// Mitsubishi GX Works2 project: 视觉检测   PLC: FX3S

PROGRAM MAIN
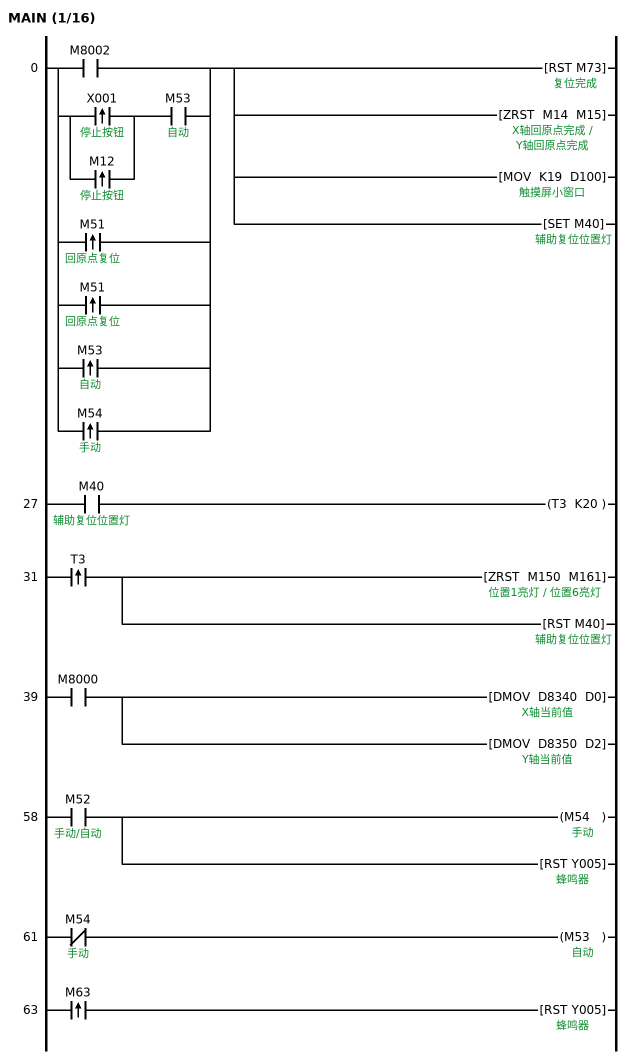
0     LD      M8002
      LDP     X001  ; 停止按钮
      ORP     M12  ; 停止按钮
      AND     M53  ; 自动
      ORB
      ORP     M51  ; 回原点复位
      ORP     M51  ; 回原点复位
      ORP     M53  ; 自动
      ORP     M54  ; 手动
      RST     M73  ; 复位完成
      ZRST    M14 M15  ; X轴回原点完成 / Y轴回原点完成
      MOV     K19 D100  ; 触摸屏小窗口
      SET     M40  ; 辅助复位位置灯
27    LD      M40  ; 辅助复位位置灯
      OUT     T3 K20
31    LDP     T3
      ZRST    M150 M161  ; 位置1亮灯 / 位置6亮灯
      RST     M40  ; 辅助复位位置灯
39    LD      M8000
      DMOV    D8340 D0  ; X轴当前值
      DMOV    D8350 D2  ; Y轴当前值
58    LD      M52  ; 手动/自动
      OUT     M54  ; 手动
      RST     Y005  ; 蜂鸣器
61    LDI     M54  ; 手动
      OUT     M53  ; 自动
63    LDP     M63
      RST     Y005  ; 蜂鸣器
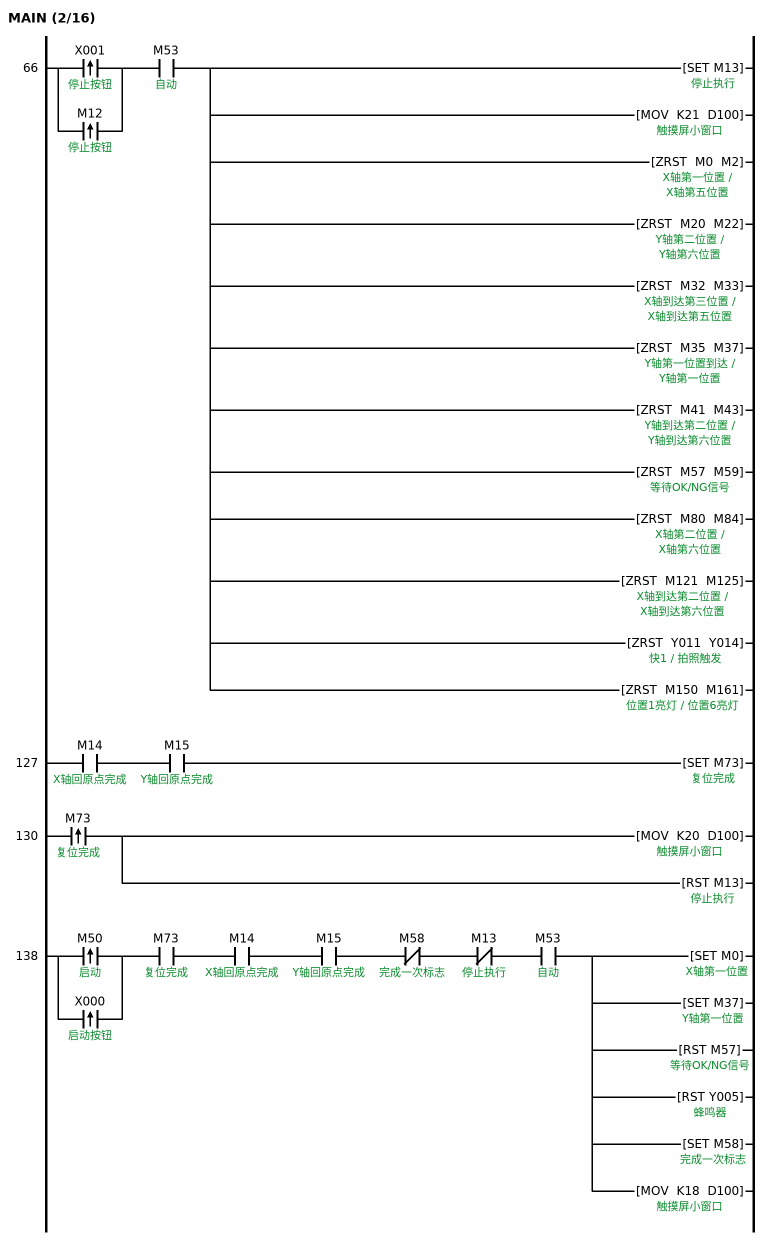
66    LDP     X001  ; 停止按钮
      ORP     M12  ; 停止按钮
      AND     M53  ; 自动
      SET     M13  ; 停止执行
      MOV     K21 D100
      ZRST    M0 M2  ; X轴第一位置 / X轴第五位置
      ZRST    M20 M22  ; Y轴第二位置 / Y轴第六位置
      ZRST    M32 M33  ; X轴到达第三位置 / X轴到达第五位置
      ZRST    M35 M37  ; Y轴第一位置到达 / Y轴第一位置
      ZRST    M41 M43  ; Y轴到达第二位置 / Y轴到达第六位置
      ZRST    M57 M59  ; 等待OK/NG信号
      ZRST    M80 M84  ; X轴第二位置 / X轴第六位置
      ZRST    M121 M125  ; X轴到达第二位置 / X轴到达第六位置
      ZRST    Y011 Y014  ; 快1 / 拍照触发
      ZRST    M150 M161
127   LD      M14  ; X轴回原点完成
      AND     M15  ; Y轴回原点完成
      SET     M73  ; 复位完成
130   LDP     M73  ; 复位完成
      MOV     K20 D100
      RST     M13  ; 停止执行
138   LDP     M50  ; 启动
      ORP     X000  ; 启动按钮
      AND     M73  ; 复位完成
      AND     M14  ; X轴回原点完成
      AND     M15  ; Y轴回原点完成
      ANI     M58  ; 完成一次标志
      ANI     M13  ; 停止执行
      AND     M53  ; 自动
      SET     M0  ; X轴第一位置
      SET     M37  ; Y轴第一位置
      RST     M57  ; 等待OK/NG信号
      RST     Y005  ; 蜂鸣器
      SET     M58  ; 完成一次标志
      MOV     K18 D100
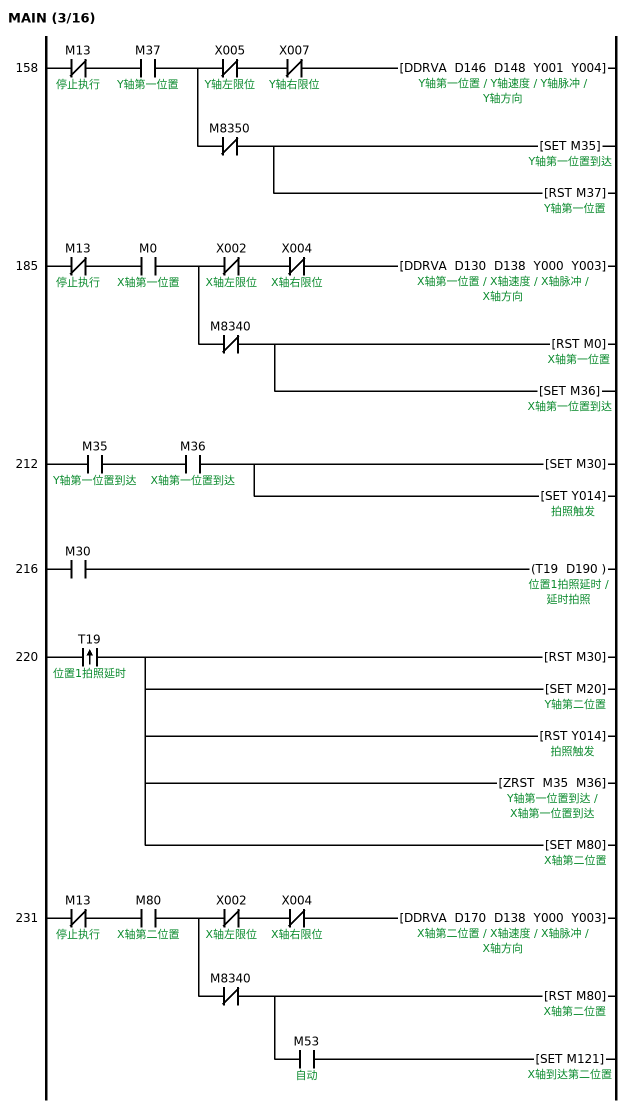
158   LDI     M13  ; 停止执行
      AND     M37  ; Y轴第一位置
      MPS
      ANI     X005  ; Y轴左限位
      ANI     X007  ; Y轴右限位
      DDRVA   D146 D148 Y001 Y004  ; Y轴第一位置 / Y轴速度 / Y轴脉冲 / Y轴方向
      MPP
      ANI     M8350
      SET     M35  ; Y轴第一位置到达
      RST     M37  ; Y轴第一位置
185   LDI     M13  ; 停止执行
      AND     M0  ; X轴第一位置
      MPS
      ANI     X002  ; X轴左限位
      ANI     X004  ; X轴右限位
      DDRVA   D130 D138 Y000 Y003  ; X轴第一位置 / X轴速度 / X轴脉冲 / X轴方向
      MPP
      ANI     M8340
      RST     M0  ; X轴第一位置
      SET     M36  ; X轴第一位置到达
212   LD      M35  ; Y轴第一位置到达
      AND     M36  ; X轴第一位置到达
      SET     M30
      SET     Y014  ; 拍照触发
216   LD      M30
      OUT     T19 D190  ; 位置1拍照延时 / 延时拍照
220   LDP     T19  ; 位置1拍照延时
      RST     M30
      SET     M20  ; Y轴第二位置
      RST     Y014  ; 拍照触发
      ZRST    M35 M36
      SET     M80  ; X轴第二位置
231   LDI     M13  ; 停止执行
      AND     M80  ; X轴第二位置
      MPS
      ANI     X002  ; X轴左限位
      ANI     X004  ; X轴右限位
      DDRVA   D170 D138 Y000 Y003  ; X轴第二位置
      MPP
      ANI     M8340
      RST     M80  ; X轴第二位置
      AND     M53  ; 自动
      SET     M121  ; X轴到达第二位置
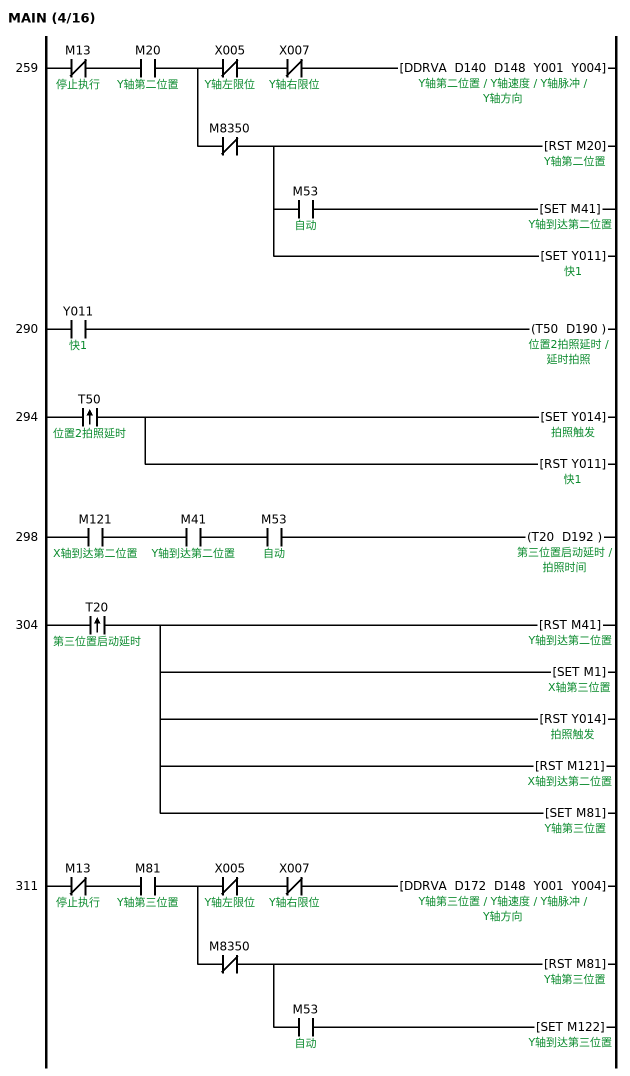
259   LDI     M13  ; 停止执行
      AND     M20  ; Y轴第二位置
      MPS
      ANI     X005  ; Y轴左限位
      ANI     X007  ; Y轴右限位
      DDRVA   D140 D148 Y001 Y004  ; Y轴第二位置
      MPP
      ANI     M8350
      RST     M20  ; Y轴第二位置
      MPS
      AND     M53  ; 自动
      SET     M41  ; Y轴到达第二位置
      MPP
      SET     Y011  ; 快1
290   LD      Y011  ; 快1
      OUT     T50 D190  ; 位置2拍照延时 / 延时拍照
294   LDP     T50  ; 位置2拍照延时
      SET     Y014  ; 拍照触发
      RST     Y011  ; 快1
298   LD      M121  ; X轴到达第二位置
      AND     M41  ; Y轴到达第二位置
      AND     M53  ; 自动
      OUT     T20 D192  ; 第三位置启动延时 / 拍照时间
304   LDP     T20  ; 第三位置启动延时
      RST     M41  ; Y轴到达第二位置
      SET     M1  ; X轴第三位置
      RST     Y014  ; 拍照触发
      RST     M121  ; X轴到达第二位置
      SET     M81  ; Y轴第三位置
311   LDI     M13  ; 停止执行
      AND     M81  ; Y轴第三位置
      MPS
      ANI     X005  ; Y轴左限位
      ANI     X007  ; Y轴右限位
      DDRVA   D172 D148 Y001 Y004  ; Y轴第三位置
      MPP
      ANI     M8350
      RST     M81  ; Y轴第三位置
      AND     M53  ; 自动
      SET     M122  ; Y轴到达第三位置
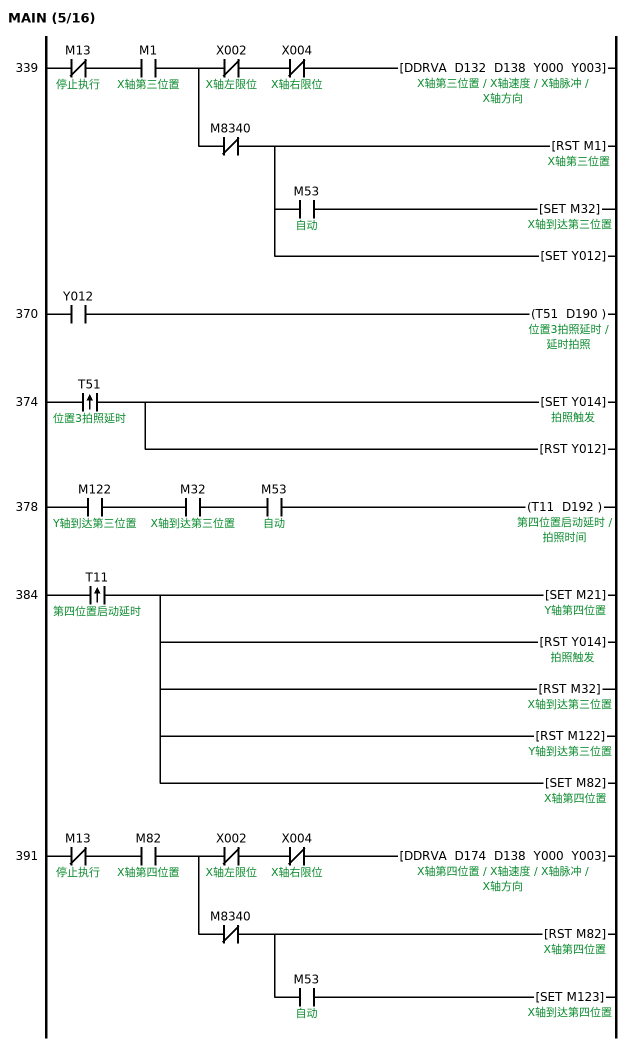
339   LDI     M13  ; 停止执行
      AND     M1  ; X轴第三位置
      MPS
      ANI     X002  ; X轴左限位
      ANI     X004  ; X轴右限位
      DDRVA   D132 D138 Y000 Y003  ; X轴第三位置
      MPP
      ANI     M8340
      RST     M1  ; X轴第三位置
      MPS
      AND     M53  ; 自动
      SET     M32  ; X轴到达第三位置
      MPP
      SET     Y012
370   LD      Y012
      OUT     T51 D190  ; 位置3拍照延时 / 延时拍照
374   LDP     T51  ; 位置3拍照延时
      SET     Y014  ; 拍照触发
      RST     Y012
378   LD      M122  ; Y轴到达第三位置
      AND     M32  ; X轴到达第三位置
      AND     M53  ; 自动
      OUT     T11 D192  ; 第四位置启动延时 / 拍照时间
384   LDP     T11  ; 第四位置启动延时
      SET     M21  ; Y轴第四位置
      RST     Y014  ; 拍照触发
      RST     M32  ; X轴到达第三位置
      RST     M122  ; Y轴到达第三位置
      SET     M82  ; X轴第四位置
391   LDI     M13  ; 停止执行
      AND     M82  ; X轴第四位置
      MPS
      ANI     X002  ; X轴左限位
      ANI     X004  ; X轴右限位
      DDRVA   D174 D138 Y000 Y003  ; X轴第四位置
      MPP
      ANI     M8340
      RST     M82  ; X轴第四位置
      AND     M53  ; 自动
      SET     M123  ; X轴到达第四位置
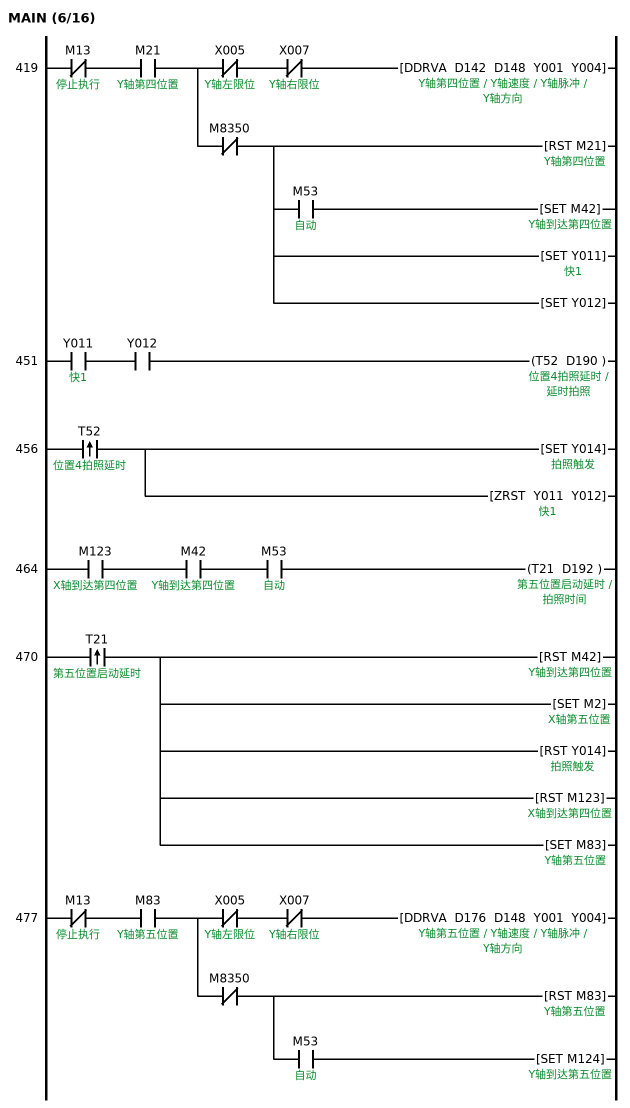
419   LDI     M13  ; 停止执行
      AND     M21  ; Y轴第四位置
      MPS
      ANI     X005  ; Y轴左限位
      ANI     X007  ; Y轴右限位
      DDRVA   D142 D148 Y001 Y004  ; Y轴第四位置
      MPP
      ANI     M8350
      RST     M21  ; Y轴第四位置
      MPS
      AND     M53  ; 自动
      SET     M42  ; Y轴到达第四位置
      MPP
      SET     Y011  ; 快1
      SET     Y012
451   LD      Y011  ; 快1
      AND     Y012
      OUT     T52 D190  ; 位置4拍照延时 / 延时拍照
456   LDP     T52  ; 位置4拍照延时
      SET     Y014  ; 拍照触发
      ZRST    Y011 Y012
464   LD      M123  ; X轴到达第四位置
      AND     M42  ; Y轴到达第四位置
      AND     M53  ; 自动
      OUT     T21 D192  ; 第五位置启动延时 / 拍照时间
470   LDP     T21  ; 第五位置启动延时
      RST     M42  ; Y轴到达第四位置
      SET     M2  ; X轴第五位置
      RST     Y014  ; 拍照触发
      RST     M123  ; X轴到达第四位置
      SET     M83  ; Y轴第五位置
477   LDI     M13  ; 停止执行
      AND     M83  ; Y轴第五位置
      MPS
      ANI     X005  ; Y轴左限位
      ANI     X007  ; Y轴右限位
      DDRVA   D176 D148 Y001 Y004  ; Y轴第五位置
      MPP
      ANI     M8350
      RST     M83  ; Y轴第五位置
      AND     M53  ; 自动
      SET     M124  ; Y轴到达第五位置
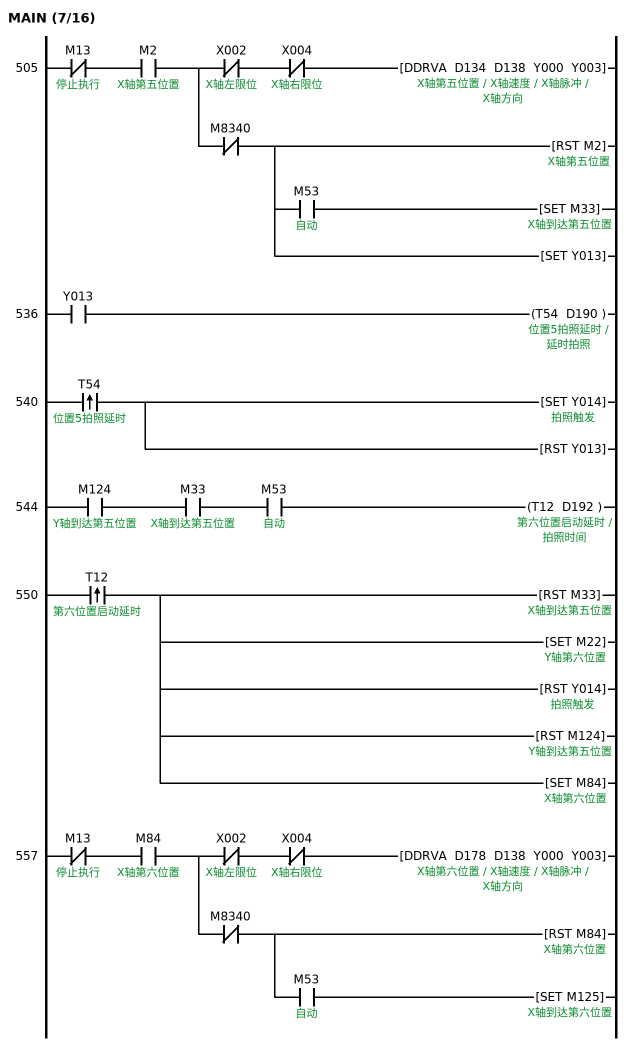
505   LDI     M13  ; 停止执行
      AND     M2  ; X轴第五位置
      MPS
      ANI     X002  ; X轴左限位
      ANI     X004  ; X轴右限位
      DDRVA   D134 D138 Y000 Y003  ; X轴第五位置
      MPP
      ANI     M8340
      RST     M2  ; X轴第五位置
      MPS
      AND     M53  ; 自动
      SET     M33  ; X轴到达第五位置
      MPP
      SET     Y013
536   LD      Y013
      OUT     T54 D190  ; 位置5拍照延时 / 延时拍照
540   LDP     T54  ; 位置5拍照延时
      SET     Y014  ; 拍照触发
      RST     Y013
544   LD      M124  ; Y轴到达第五位置
      AND     M33  ; X轴到达第五位置
      AND     M53  ; 自动
      OUT     T12 D192  ; 第六位置启动延时 / 拍照时间
550   LDP     T12  ; 第六位置启动延时
      RST     M33  ; X轴到达第五位置
      SET     M22  ; Y轴第六位置
      RST     Y014  ; 拍照触发
      RST     M124  ; Y轴到达第五位置
      SET     M84  ; X轴第六位置
557   LDI     M13  ; 停止执行
      AND     M84  ; X轴第六位置
      MPS
      ANI     X002  ; X轴左限位
      ANI     X004  ; X轴右限位
      DDRVA   D178 D138 Y000 Y003  ; X轴第六位置
      MPP
      ANI     M8340
      RST     M84  ; X轴第六位置
      AND     M53  ; 自动
      SET     M125  ; X轴到达第六位置
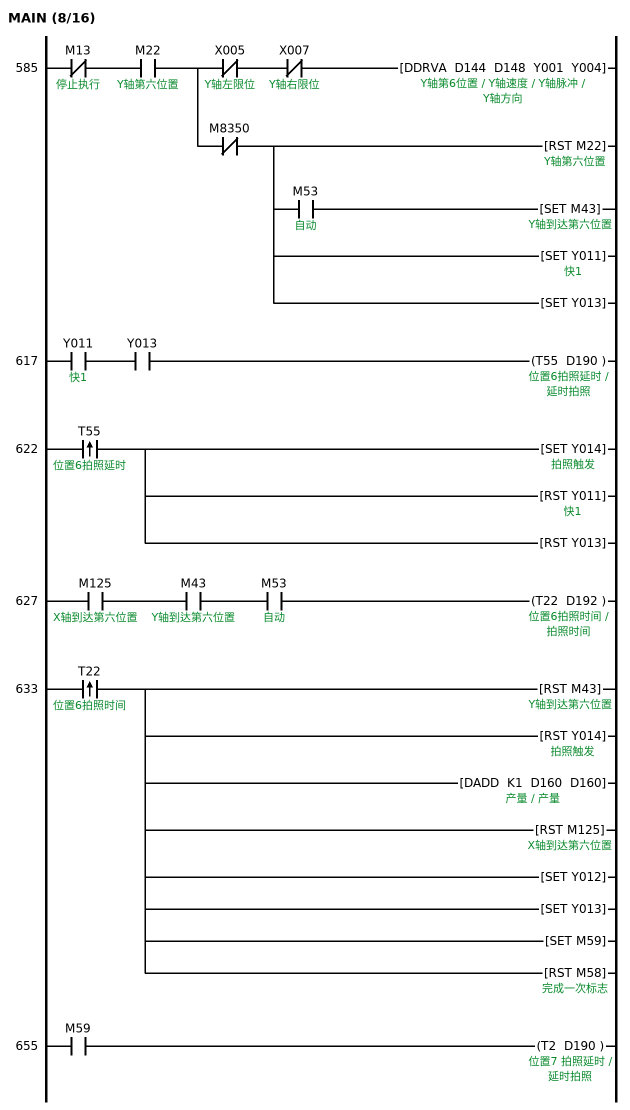
585   LDI     M13  ; 停止执行
      AND     M22  ; Y轴第六位置
      MPS
      ANI     X005  ; Y轴左限位
      ANI     X007  ; Y轴右限位
      DDRVA   D144 D148 Y001 Y004  ; Y轴第6位置
      MPP
      ANI     M8350
      RST     M22  ; Y轴第六位置
      MPS
      AND     M53  ; 自动
      SET     M43  ; Y轴到达第六位置
      MPP
      SET     Y011  ; 快1
      SET     Y013
617   LD      Y011  ; 快1
      AND     Y013
      OUT     T55 D190  ; 位置6拍照延时 / 延时拍照
622   LDP     T55  ; 位置6拍照延时
      SET     Y014  ; 拍照触发
      RST     Y011  ; 快1
      RST     Y013
627   LD      M125  ; X轴到达第六位置
      AND     M43  ; Y轴到达第六位置
      AND     M53  ; 自动
      OUT     T22 D192  ; 位置6拍照时间 / 拍照时间
633   LDP     T22  ; 位置6拍照时间
      RST     M43  ; Y轴到达第六位置
      RST     Y014  ; 拍照触发
      DADD    K1 D160 D160  ; 产量
      RST     M125  ; X轴到达第六位置
      SET     Y012
      SET     Y013
      SET     M59
      RST     M58  ; 完成一次标志
655   LD      M59
      OUT     T2 D190  ; 位置7 拍照延时 / 延时拍照
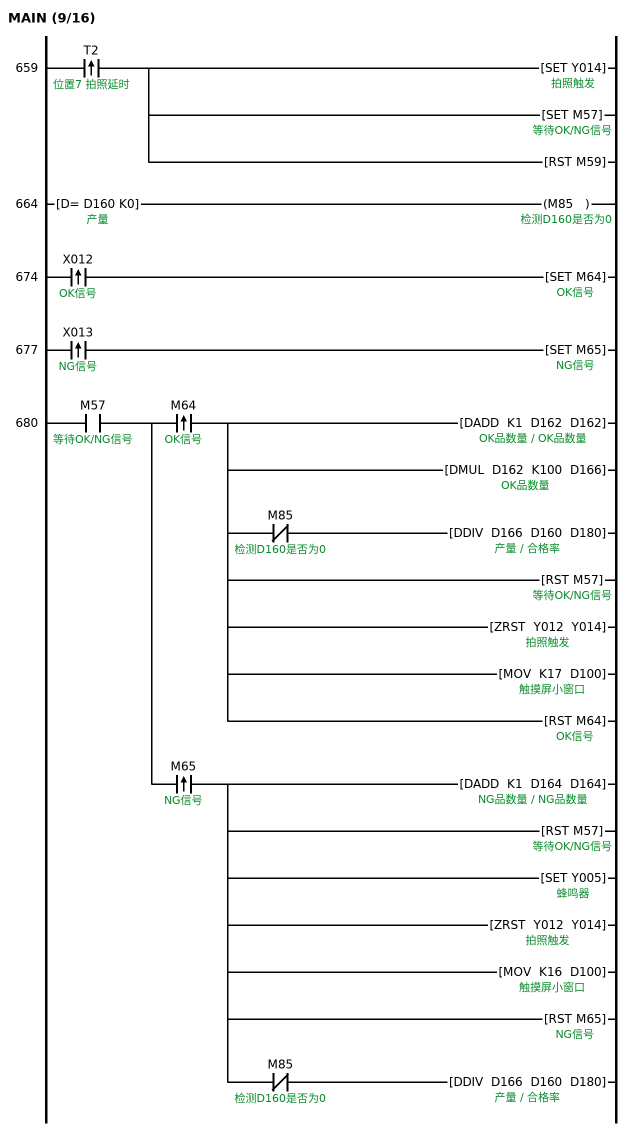
659   LDP     T2  ; 位置7 拍照延时
      SET     Y014  ; 拍照触发
      SET     M57  ; 等待OK/NG信号
      RST     M59
664   LDD=    D160 K0  ; 产量
      OUT     M85  ; 检测D160是否为0
674   LDP     X012  ; OK信号
      SET     M64  ; OK信号
677   LDP     X013  ; NG信号
      SET     M65  ; NG信号
680   LD      M57  ; 等待OK/NG信号
      MPS
      ANDP    M64  ; OK信号
      DADD    K1 D162 D162  ; OK品数量
      DMUL    D162 K100 D166
      MPS
      ANI     M85  ; 检测D160是否为0
      DDIV    D166 D160 D180  ; 合格率
      MPP
      RST     M57  ; 等待OK/NG信号
      ZRST    Y012 Y014
      MOV     K17 D100
      RST     M64  ; OK信号
      MPP
      ANDP    M65  ; NG信号
      DADD    K1 D164 D164  ; NG品数量
      RST     M57  ; 等待OK/NG信号
      SET     Y005  ; 蜂鸣器
      ZRST    Y012 Y014
      MOV     K16 D100
      RST     M65  ; NG信号
      ANI     M85  ; 检测D160是否为0
      DDIV    D166 D160 D180
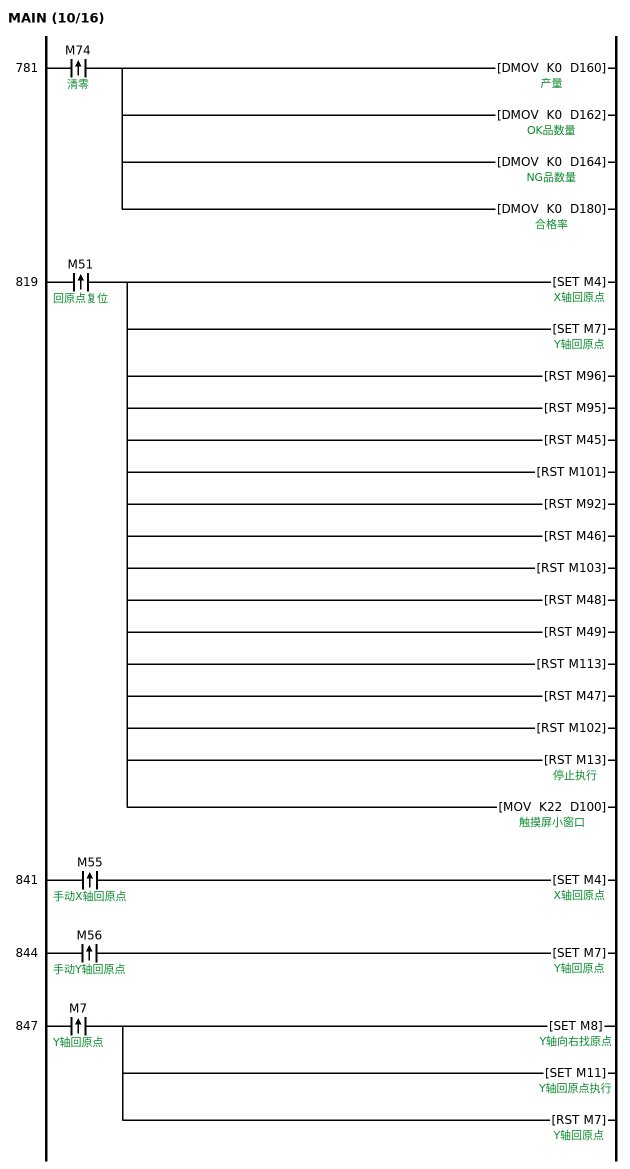
781   LDP     M74  ; 清零
      DMOV    K0 D160
      DMOV    K0 D162
      DMOV    K0 D164
      DMOV    K0 D180
819   LDP     M51  ; 回原点复位
      SET     M4  ; X轴回原点
      SET     M7  ; Y轴回原点
      RST     M96
      RST     M95
      RST     M45
      RST     M101
      RST     M92
      RST     M46
      RST     M103
      RST     M48
      RST     M49
      RST     M113
      RST     M47
      RST     M102
      RST     M13  ; 停止执行
      MOV     K22 D100
841   LDP     M55  ; 手动X轴回原点
      SET     M4  ; X轴回原点
844   LDP     M56  ; 手动Y轴回原点
      SET     M7  ; Y轴回原点
847   LDP     M7  ; Y轴回原点
      SET     M8  ; Y轴向右找原点
      SET     M11  ; Y轴回原点执行
      RST     M7  ; Y轴回原点
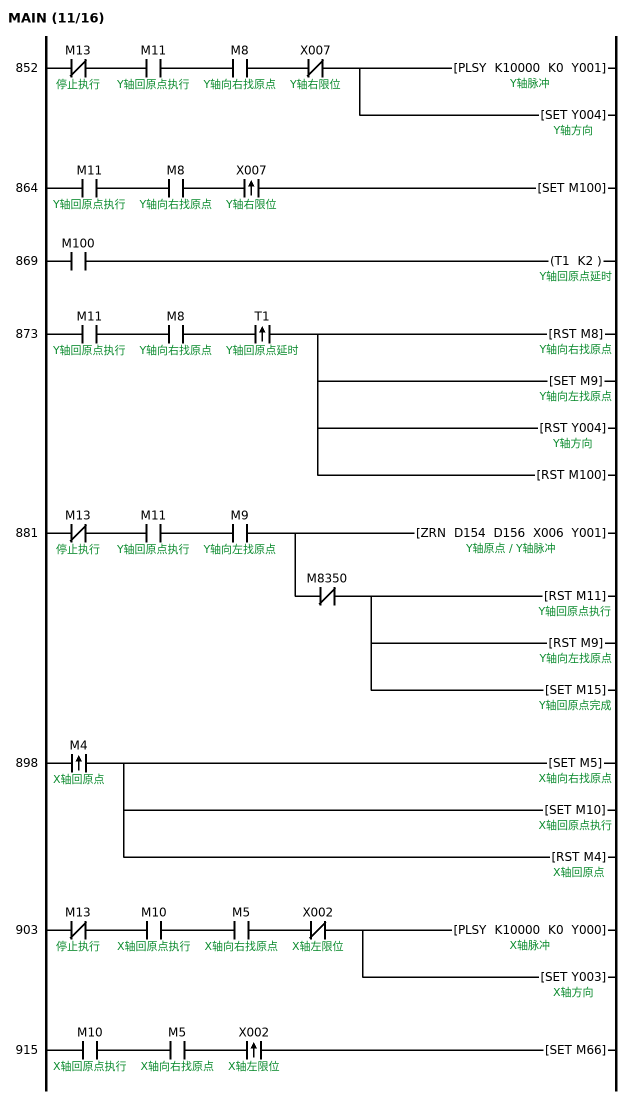
852   LDI     M13  ; 停止执行
      AND     M11  ; Y轴回原点执行
      AND     M8  ; Y轴向右找原点
      ANI     X007  ; Y轴右限位
      PLSY    K10000 K0 Y001  ; Y轴脉冲
      SET     Y004  ; Y轴方向
864   LD      M11  ; Y轴回原点执行
      AND     M8  ; Y轴向右找原点
      ANDP    X007  ; Y轴右限位
      SET     M100
869   LD      M100
      OUT     T1 K2  ; Y轴回原点延时
873   LD      M11  ; Y轴回原点执行
      AND     M8  ; Y轴向右找原点
      ANDP    T1  ; Y轴回原点延时
      RST     M8  ; Y轴向右找原点
      SET     M9  ; Y轴向左找原点
      RST     Y004  ; Y轴方向
      RST     M100
881   LDI     M13  ; 停止执行
      AND     M11  ; Y轴回原点执行
      AND     M9  ; Y轴向左找原点
      ZRN     D154 D156 X006 Y001  ; Y轴原点
      ANI     M8350
      RST     M11  ; Y轴回原点执行
      RST     M9  ; Y轴向左找原点
      SET     M15  ; Y轴回原点完成
898   LDP     M4  ; X轴回原点
      SET     M5  ; X轴向右找原点
      SET     M10  ; X轴回原点执行
      RST     M4  ; X轴回原点
903   LDI     M13  ; 停止执行
      AND     M10  ; X轴回原点执行
      AND     M5  ; X轴向右找原点
      ANI     X002  ; X轴左限位
      PLSY    K10000 K0 Y000  ; X轴脉冲
      SET     Y003  ; X轴方向
915   LD      M10  ; X轴回原点执行
      AND     M5  ; X轴向右找原点
      ANDP    X002  ; X轴左限位
      SET     M66
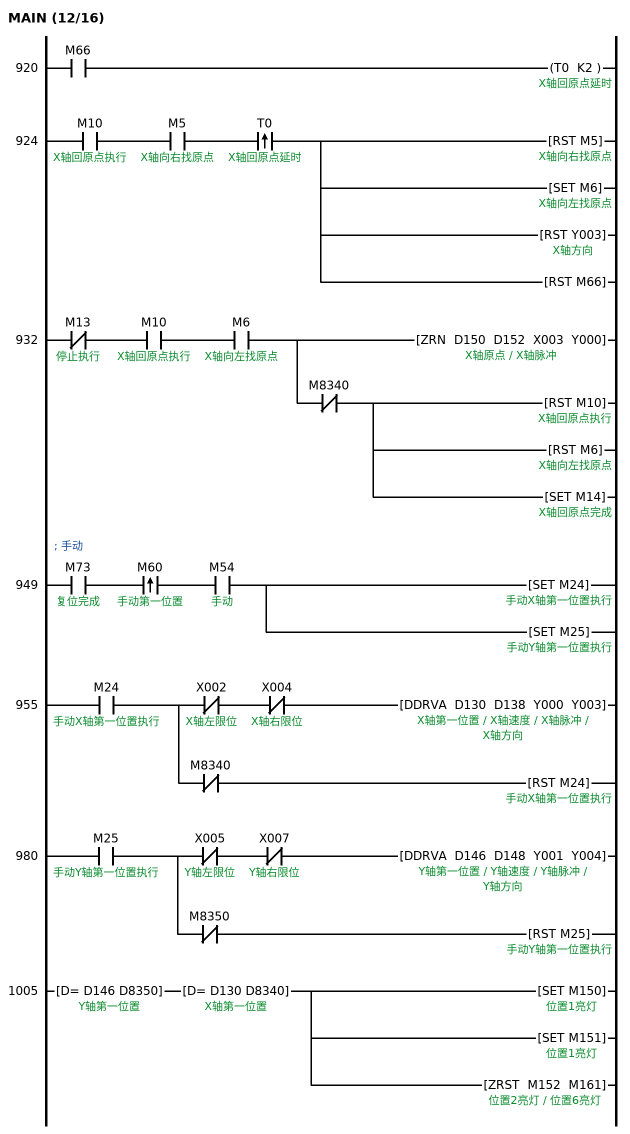
920   LD      M66
      OUT     T0 K2  ; X轴回原点延时
924   LD      M10  ; X轴回原点执行
      AND     M5  ; X轴向右找原点
      ANDP    T0  ; X轴回原点延时
      RST     M5  ; X轴向右找原点
      SET     M6  ; X轴向左找原点
      RST     Y003  ; X轴方向
      RST     M66
932   LDI     M13  ; 停止执行
      AND     M10  ; X轴回原点执行
      AND     M6  ; X轴向左找原点
      ZRN     D150 D152 X003 Y000  ; X轴原点
      ANI     M8340
      RST     M10  ; X轴回原点执行
      RST     M6  ; X轴向左找原点
      SET     M14  ; X轴回原点完成
; 手动
949   LD      M73  ; 复位完成
      ANDP    M60  ; 手动第一位置
      AND     M54  ; 手动
      SET     M24  ; 手动X轴第一位置执行
      SET     M25  ; 手动Y轴第一位置执行
955   LD      M24  ; 手动X轴第一位置执行
      MPS
      ANI     X002  ; X轴左限位
      ANI     X004  ; X轴右限位
      DDRVA   D130 D138 Y000 Y003
      MPP
      ANI     M8340
      RST     M24  ; 手动X轴第一位置执行
980   LD      M25  ; 手动Y轴第一位置执行
      MPS
      ANI     X005  ; Y轴左限位
      ANI     X007  ; Y轴右限位
      DDRVA   D146 D148 Y001 Y004
      MPP
      ANI     M8350
      RST     M25  ; 手动Y轴第一位置执行
1005  LDD=    D146 D8350  ; Y轴第一位置
      ANDD=   D130 D8340  ; X轴第一位置
      SET     M150  ; 位置1亮灯
      SET     M151  ; 位置1亮灯
      ZRST    M152 M161  ; 位置2亮灯
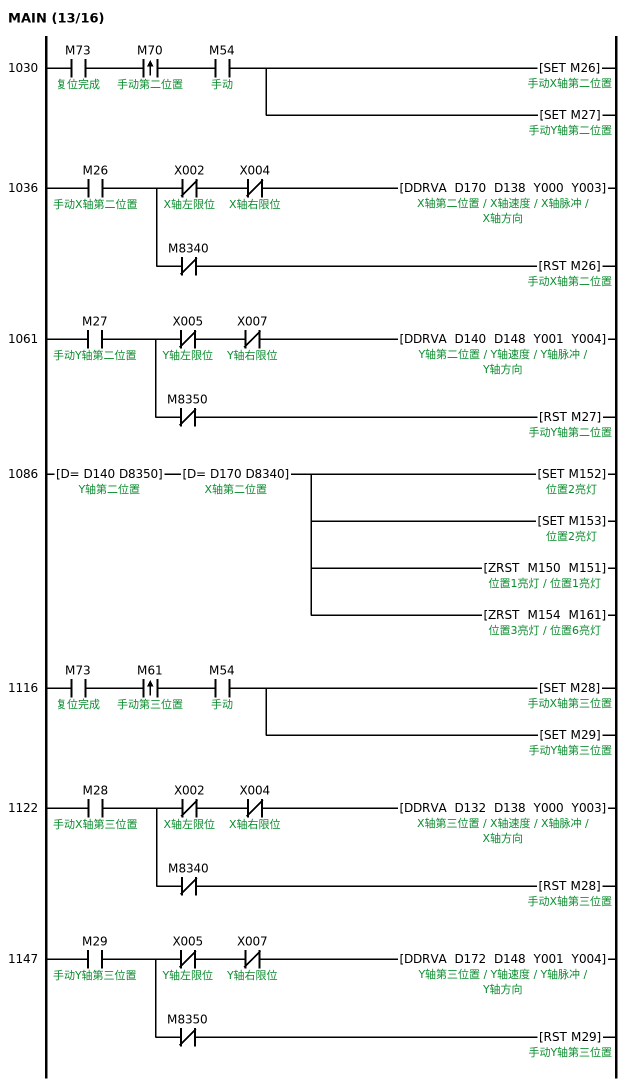
1030  LD      M73  ; 复位完成
      ANDP    M70  ; 手动第二位置
      AND     M54  ; 手动
      SET     M26  ; 手动X轴第二位置
      SET     M27  ; 手动Y轴第二位置
1036  LD      M26  ; 手动X轴第二位置
      MPS
      ANI     X002  ; X轴左限位
      ANI     X004  ; X轴右限位
      DDRVA   D170 D138 Y000 Y003
      MPP
      ANI     M8340
      RST     M26  ; 手动X轴第二位置
1061  LD      M27  ; 手动Y轴第二位置
      MPS
      ANI     X005  ; Y轴左限位
      ANI     X007  ; Y轴右限位
      DDRVA   D140 D148 Y001 Y004
      MPP
      ANI     M8350
      RST     M27  ; 手动Y轴第二位置
1086  LDD=    D140 D8350  ; Y轴第二位置
      ANDD=   D170 D8340  ; X轴第二位置
      SET     M152  ; 位置2亮灯
      SET     M153  ; 位置2亮灯
      ZRST    M150 M151
      ZRST    M154 M161  ; 位置3亮灯
1116  LD      M73  ; 复位完成
      ANDP    M61  ; 手动第三位置
      AND     M54  ; 手动
      SET     M28  ; 手动X轴第三位置
      SET     M29  ; 手动Y轴第三位置
1122  LD      M28  ; 手动X轴第三位置
      MPS
      ANI     X002  ; X轴左限位
      ANI     X004  ; X轴右限位
      DDRVA   D132 D138 Y000 Y003
      MPP
      ANI     M8340
      RST     M28  ; 手动X轴第三位置
1147  LD      M29  ; 手动Y轴第三位置
      MPS
      ANI     X005  ; Y轴左限位
      ANI     X007  ; Y轴右限位
      DDRVA   D172 D148 Y001 Y004
      MPP
      ANI     M8350
      RST     M29  ; 手动Y轴第三位置
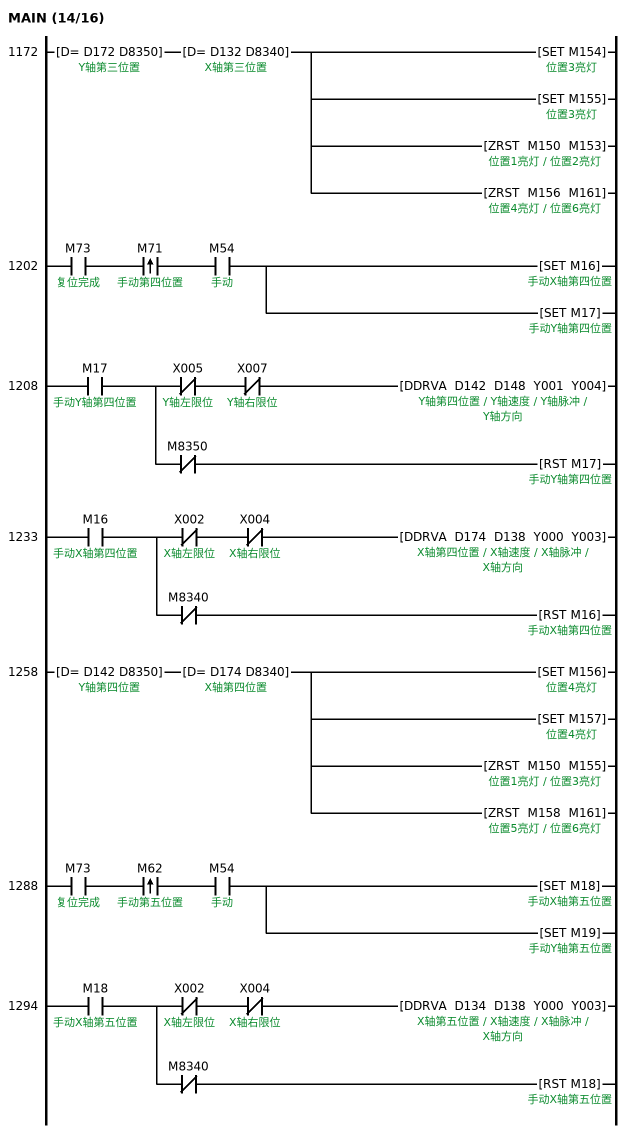
1172  LDD=    D172 D8350  ; Y轴第三位置
      ANDD=   D132 D8340  ; X轴第三位置
      SET     M154  ; 位置3亮灯
      SET     M155  ; 位置3亮灯
      ZRST    M150 M153
      ZRST    M156 M161  ; 位置4亮灯
1202  LD      M73  ; 复位完成
      ANDP    M71  ; 手动第四位置
      AND     M54  ; 手动
      SET     M16  ; 手动X轴第四位置
      SET     M17  ; 手动Y轴第四位置
1208  LD      M17  ; 手动Y轴第四位置
      MPS
      ANI     X005  ; Y轴左限位
      ANI     X007  ; Y轴右限位
      DDRVA   D142 D148 Y001 Y004
      MPP
      ANI     M8350
      RST     M17  ; 手动Y轴第四位置
1233  LD      M16  ; 手动X轴第四位置
      MPS
      ANI     X002  ; X轴左限位
      ANI     X004  ; X轴右限位
      DDRVA   D174 D138 Y000 Y003
      MPP
      ANI     M8340
      RST     M16  ; 手动X轴第四位置
1258  LDD=    D142 D8350  ; Y轴第四位置
      ANDD=   D174 D8340  ; X轴第四位置
      SET     M156  ; 位置4亮灯
      SET     M157  ; 位置4亮灯
      ZRST    M150 M155
      ZRST    M158 M161  ; 位置5亮灯
1288  LD      M73  ; 复位完成
      ANDP    M62  ; 手动第五位置
      AND     M54  ; 手动
      SET     M18  ; 手动X轴第五位置
      SET     M19  ; 手动Y轴第五位置
1294  LD      M18  ; 手动X轴第五位置
      MPS
      ANI     X002  ; X轴左限位
      ANI     X004  ; X轴右限位
      DDRVA   D134 D138 Y000 Y003
      MPP
      ANI     M8340
      RST     M18  ; 手动X轴第五位置
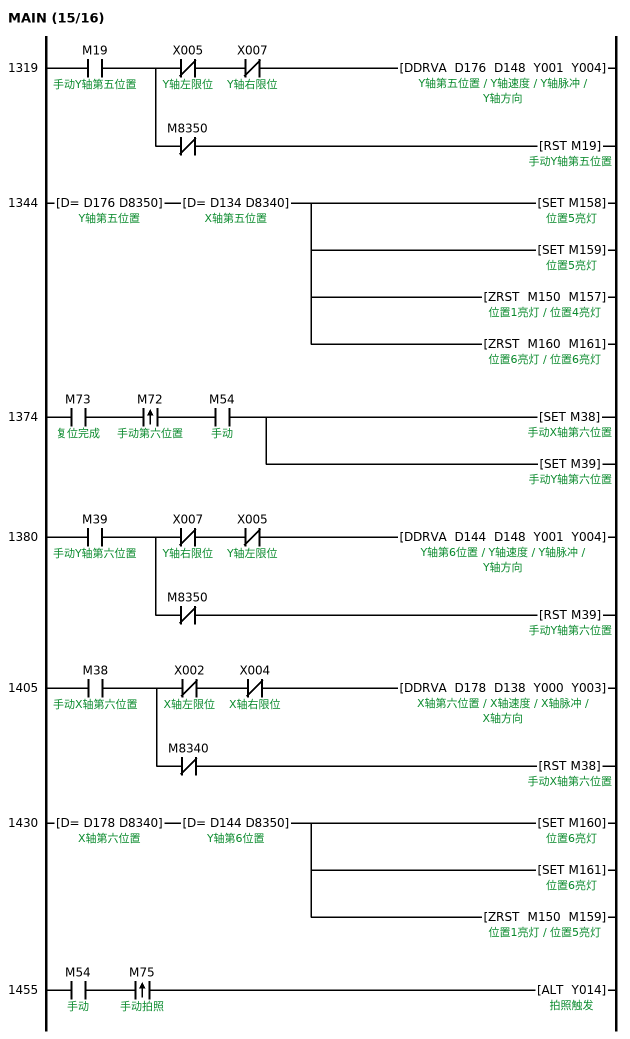
1319  LD      M19  ; 手动Y轴第五位置
      MPS
      ANI     X005  ; Y轴左限位
      ANI     X007  ; Y轴右限位
      DDRVA   D176 D148 Y001 Y004
      MPP
      ANI     M8350
      RST     M19  ; 手动Y轴第五位置
1344  LDD=    D176 D8350  ; Y轴第五位置
      ANDD=   D134 D8340  ; X轴第五位置
      SET     M158  ; 位置5亮灯
      SET     M159  ; 位置5亮灯
      ZRST    M150 M157
      ZRST    M160 M161  ; 位置6亮灯
1374  LD      M73  ; 复位完成
      ANDP    M72  ; 手动第六位置
      AND     M54  ; 手动
      SET     M38  ; 手动X轴第六位置
      SET     M39  ; 手动Y轴第六位置
1380  LD      M39  ; 手动Y轴第六位置
      MPS
      ANI     X007  ; Y轴右限位
      ANI     X005  ; Y轴左限位
      DDRVA   D144 D148 Y001 Y004
      MPP
      ANI     M8350
      RST     M39  ; 手动Y轴第六位置
1405  LD      M38  ; 手动X轴第六位置
      MPS
      ANI     X002  ; X轴左限位
      ANI     X004  ; X轴右限位
      DDRVA   D178 D138 Y000 Y003
      MPP
      ANI     M8340
      RST     M38  ; 手动X轴第六位置
1430  LDD=    D178 D8340  ; X轴第六位置
      ANDD=   D144 D8350  ; Y轴第6位置
      SET     M160  ; 位置6亮灯
      SET     M161  ; 位置6亮灯
      ZRST    M150 M159
1455  LD      M54  ; 手动
      ANDP    M75  ; 手动拍照
      ALT     Y014
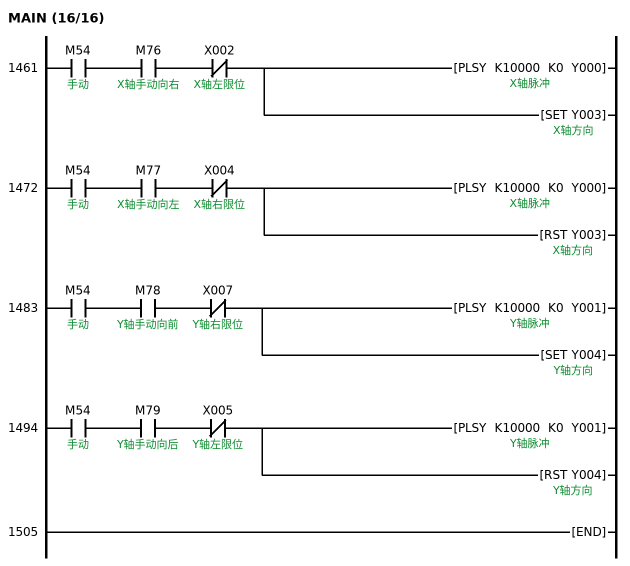
1461  LD      M54  ; 手动
      AND     M76  ; X轴手动向右
      ANI     X002  ; X轴左限位
      PLSY    K10000 K0 Y000  ; X轴脉冲
      SET     Y003  ; X轴方向
1472  LD      M54  ; 手动
      AND     M77  ; X轴手动向左
      ANI     X004  ; X轴右限位
      PLSY    K10000 K0 Y000  ; X轴脉冲
      RST     Y003  ; X轴方向
1483  LD      M54  ; 手动
      AND     M78  ; Y轴手动向前
      ANI     X007  ; Y轴右限位
      PLSY    K10000 K0 Y001  ; Y轴脉冲
      SET     Y004  ; Y轴方向
1494  LD      M54  ; 手动
      AND     M79  ; Y轴手动向后
      ANI     X005  ; Y轴左限位
      PLSY    K10000 K0 Y001  ; Y轴脉冲
      RST     Y004  ; Y轴方向
1505  END
END_PROGRAM

// device comments not shown above
Y006  ; 黄灯
Y007  ; 绿灯
M3  ; 轴1第四位置
M23  ; Y轴第四位置
M90  ; 轴1原点完成
M91  ; 轴2原点完成
T10  ; 轴1第二位置启动延时
